{region '#Template'}
	{attribute 'Category' := 'Universal'}
	{attribute 'Version' := '0.0.1.0'}
	{attribute 'Tags' := 'Universal, Control, Hysteresis'}
	{attribute 'Description' := 'Hysterese	// Hysteresis'}
{endregion}
FUNCTION_BLOCK FB_BA_Hys_21 EXTENDS FB_BA_View
VAR_INPUT
	bEn 					: BOOL := TRUE;	
	fIn						: REAL;
END_VAR
VAR_OUTPUT
	bDst					: BOOL;
END_VAR
VAR_INPUT CONSTANT
	HysPreAlarmOn			: FB_BA_AV_Op;		
	HysPreAlarmOff			: FB_BA_AV_Op;		
	HysMainAlarmOn			: FB_BA_AV_Op;		
	HysMainAlarmOff			: FB_BA_AV_Op;	
	DstPreAlarm				: FB_BA_BV;
	DstMainAlarm			: FB_BA_BV;
END_VAR
VAR
	HysPreAlarm				: FB_BA_Swi2P;
	HysMainAlarm			: FB_BA_Swi2P;
END_VAR

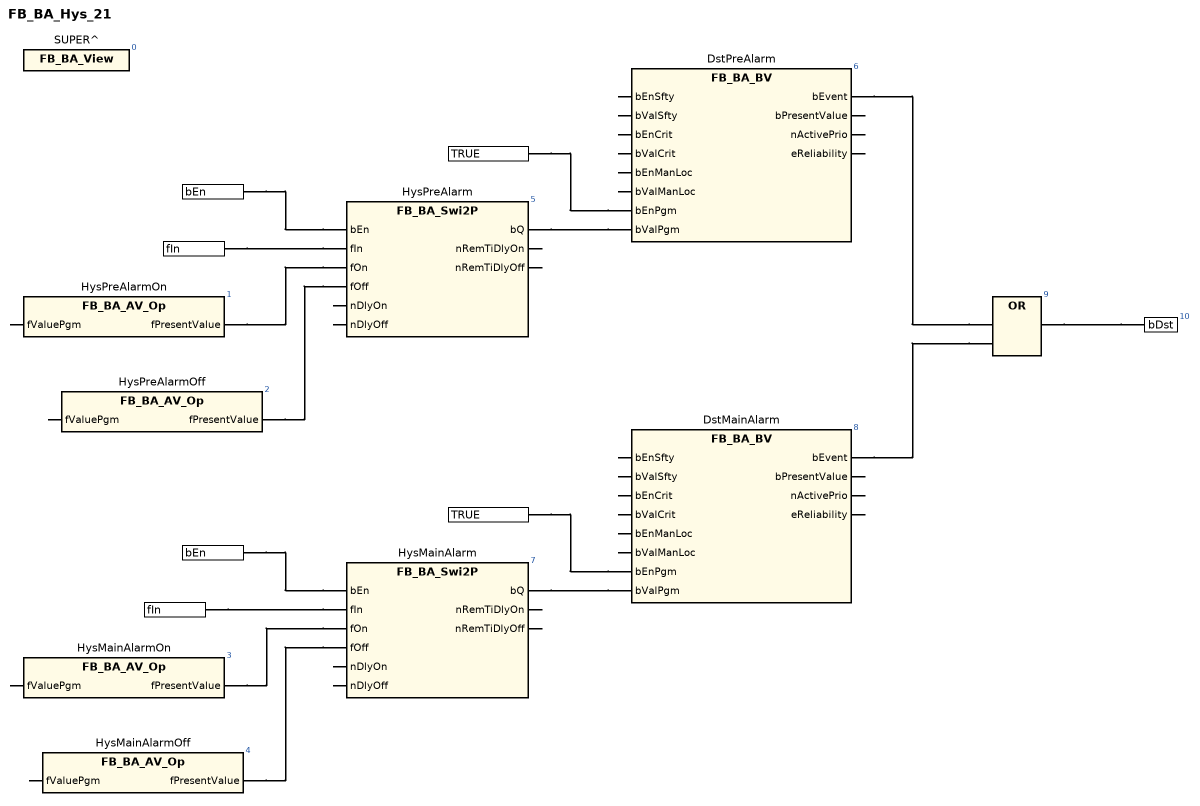
SUPER^(); // FB_BA_View
HysPreAlarmOn(); // FB_BA_AV_Op
HysPreAlarmOff(); // FB_BA_AV_Op
HysMainAlarmOn(); // FB_BA_AV_Op
HysMainAlarmOff(); // FB_BA_AV_Op
HysPreAlarm(bEn := bEn, fIn := fIn, fOn := HysPreAlarmOn.fPresentValue, fOff := HysPreAlarmOff.fPresentValue); // FB_BA_Swi2P
DstPreAlarm(bEnPgm := TRUE, bValPgm := HysPreAlarm.bQ); // FB_BA_BV
HysMainAlarm(
    bEn := bEn,
    fIn := fIn,
    fOn := HysMainAlarmOn.fPresentValue,
    fOff := HysMainAlarmOff.fPresentValue); // FB_BA_Swi2P
DstMainAlarm(bEnPgm := TRUE, bValPgm := HysMainAlarm.bQ); // FB_BA_BV
bDst := DstPreAlarm.bEvent OR DstMainAlarm.bEvent;

METHOD FB_init : BOOL
VAR_INPUT
	bInitRetains : BOOL; // if TRUE, the retain variables are initialized (warm start / cold start)
	bInCopyCode : BOOL;  // if TRUE, the instance afterwards gets moved into the copy code (online change)
END_VAR
HysPreAlarmOn.iParent						:= THIS^;
HysPreAlarmOn.iLabel						:= LblUniControl.Hysteresis_PreAlarmLimitMAX;	 
HysPreAlarmOn.sObjectName					:= '{Idx=01}';	
HysPreAlarmOn.eUnit							:= E_BA_Unit.ePressure_Pascals;							 	 
HysPreAlarmOn.fValueRm						:= 200;			
HysPreAlarmOn.fCOVIncrement					:= BA2_Param.fDefCOVIncrement;		

HysPreAlarmOff.iParent						:= THIS^;
HysPreAlarmOff.iLabel						:= LblUniControl.Hysteresis_PreAlarmLimitMIN;	 
HysPreAlarmOff.sObjectName					:= '{Idx=01}';	
HysPreAlarmOff.eUnit						:= E_BA_Unit.ePressure_Pascals;							 	 
HysPreAlarmOff.fValueRm						:= 150;			
HysPreAlarmOff.fCOVIncrement				:= BA2_Param.fDefCOVIncrement;		
							
HysMainAlarmOn.iParent						:= THIS^;
HysMainAlarmOn.iLabel						:= LblUniControl.Hysteresis_MainAlarmLimitMAX; 
HysMainAlarmOn.sObjectName					:= '{Idx=02}';								 	 
HysMainAlarmOn.eUnit						:= E_BA_Unit.ePressure_Pascals;
HysMainAlarmOn.fValueRm						:= 350;			
HysMainAlarmOn.fCOVIncrement				:= BA2_Param.fDefCOVIncrement;		
							
HysMainAlarmOff.iParent						:= THIS^;
HysMainAlarmOff.iLabel						:= LblUniControl.Hysteresis_MainAlarmLimitMIN; 
HysMainAlarmOff.sObjectName					:= '{Idx=02}';								 	 
HysMainAlarmOff.eUnit						:= E_BA_Unit.ePressure_Pascals;
HysMainAlarmOff.fValueRm					:= 300;			
HysMainAlarmOff.fCOVIncrement				:= BA2_Param.fDefCOVIncrement;		

DstPreAlarm.iParent							:= THIS^;
DstPreAlarm.iLabel							:= LblUniControl.Hysteresis_PreAlarmFault;			
DstPreAlarm.sObjectName						:= '{Idx=01}';	
DstPreAlarm.bEnOutOfService					:= FALSE;
DstPreAlarm.sActiveText 					:= Texts.txtMaintenace;
DstPreAlarm.sInactiveText 					:= Texts.txtNormal;
DstPreAlarm.nStateChangeCount				:= 0;
DstPreAlarm.nActiveTimeElapsed				:= 0;
DstPreAlarm.nMinimumOnTime					:= 0;
DstPreAlarm.nMinimumOffTime					:= 0;
DstPreAlarm.bEnManualRm						:= FALSE;	//	Priority  8	
DstPreAlarm.bValManualRm					:= FALSE;	//	Priority  8
DstPreAlarm.bDefaultValue					:= FALSE;
DstPreAlarm.nEventClassID					:= EventClasses.MaintenanceSimple;
DstPreAlarm.stTimeDelay.nToNormal			:= BA2_Param.nDefTimeDelay_ToNormal;
DstPreAlarm.stTimeDelay.nToAbnormal			:= BA2_Param.nDefTimeDelay_ToAbnormal;
DstPreAlarm.bAlarmValue						:= TRUE;
DstPreAlarm.bAcknowledgeRm					:= FALSE;		
DstPreAlarm.aEventTransitionText[1]			:= Texts.txtDisturb;
DstPreAlarm.aEventTransitionText[2]			:= Texts.txtNone;
DstPreAlarm.aEventTransitionText[3]			:= Texts.txtNormal;
DstPreAlarm.bEventDetectionEnable			:= TRUE;
DstPreAlarm.eEnPlantLock					:= E_BA_LockPriority.eNoLock;	

DstMainAlarm.iParent						:= THIS^;
DstMainAlarm.iLabel							:= LblUniControl.Hysteresis_MainAlarmFault;			
DstMainAlarm.sObjectName					:= '{Idx=02}';	
DstMainAlarm.bEnOutOfService				:= FALSE;
DstMainAlarm.sActiveText 					:= Texts.txtTriggered;
DstMainAlarm.sInactiveText 					:= Texts.txtNormal;
DstMainAlarm.nStateChangeCount				:= 0;
DstMainAlarm.nActiveTimeElapsed				:= 0;
DstMainAlarm.nMinimumOnTime					:= 0;
DstMainAlarm.nMinimumOffTime				:= 0;
DstMainAlarm.bEnManualRm					:= FALSE;	//	Priority  8	
DstMainAlarm.bValManualRm					:= FALSE;	//	Priority  8
DstMainAlarm.bDefaultValue					:= FALSE;
DstMainAlarm.nEventClassID					:= EventClasses.AlarmTechnicalExtended;
DstMainAlarm.stTimeDelay.nToNormal			:= BA2_Param.nDefTimeDelay_ToNormal;
DstMainAlarm.stTimeDelay.nToAbnormal		:= BA2_Param.nDefTimeDelay_ToAbnormal;
DstMainAlarm.bAlarmValue					:= TRUE;
DstMainAlarm.bAcknowledgeRm					:= FALSE;		
DstMainAlarm.aEventTransitionText[1]		:= Texts.txtTriggered;
DstMainAlarm.aEventTransitionText[2]		:= Texts.txtError;
DstMainAlarm.aEventTransitionText[3]		:= Texts.txtNormal;
DstMainAlarm.bEventDetectionEnable			:= TRUE;
DstMainAlarm.eEnPlantLock					:= E_BA_LockPriority.eNoLock;
END_METHOD

END_FUNCTION_BLOCK

(* stored: Version 1.1.0.1, ProductVersion 3.1.4024.6
   POU FB_BA_Hys_21: Id {a495cf77-b79e-4333-ace5-202f1a9b862b}, SpecialFunc None
   Method FB_init: Id {708c9e99-f714-465f-bb1f-19e526ec0016} *)
